INTERFACE ITF_ControlElement_1 EXTENDS ITF_BaseControlElement

END_INTERFACE

(* stored: Version 1.1.0.1, ProductVersion 3.1.4024.15
   Itf ITF_ControlElement_1: Id {16db250a-4be8-49f7-ab8b-5e7acb82e030} *)
